FUNCTION F_HV_ILK : BOOL
VAR_INPUT
	IG	:	ST_VG; // Gauge used for interlocking the high voltage supply 
	HV	:	ST_HV; // Structure representing HV control
END_VAR
VAR
END_VAR

F_HV_ILK := ((IG.xPRESS_OK = TRUE)
			AND (IG.rPRESS < HV.rPRO_SP));

END_FUNCTION

(* stored: Version 1.1.0.1, ProductVersion 3.1.4024.2
   POU F_HV_ILK: Id {93ea2e20-5fc5-4962-9409-abe8b95bf005}, SpecialFunc None *)
